INTERFACE PUBLIC RelativeMoveBuilder EXTENDS __System.IQueryInterface

METHOD PUBLIC Acceleration : RelativeMoveBuilder
VAR_INPUT
	value : LREAL;
END_VAR
END_METHOD

METHOD PUBLIC BufferMode : RelativeMoveBuilder
VAR_INPUT
	mode : MotionBufferMode;
END_VAR
END_METHOD

METHOD PUBLIC BuildMoveAdditiveCommand : MotionCommand
VAR_INPUT
	axis : Axis;
END_VAR
END_METHOD

METHOD PUBLIC BuildMoveRelativeCommand : MotionCommand
VAR_INPUT
	axis : Axis;
END_VAR
END_METHOD

METHOD PUBLIC Deceleration : RelativeMoveBuilder
VAR_INPUT
	value : LREAL;
END_VAR
END_METHOD

METHOD PUBLIC Distance : RelativeMoveBuilder
VAR_INPUT
	value : LREAL;
END_VAR
END_METHOD

METHOD PUBLIC Jerk : RelativeMoveBuilder
VAR_INPUT
	value : LREAL;
END_VAR
END_METHOD

METHOD PUBLIC Velocity : RelativeMoveBuilder
VAR_INPUT
	value : LREAL;
END_VAR
END_METHOD

END_INTERFACE

(* stored: Version 1.1.0.1
   Itf RelativeMoveBuilder: Id {bddc8931-0c19-0eb2-24a5-b0ff1c07fd66}
   Folder Builders: Id {6daf0ca8-bdaf-495b-8bb7-ee7370bef123}
   Folder PropertySetters: Id {1d69e98f-87ac-4f4f-9b60-ecee3ad0fec2}
   Method Acceleration: Id {6f259ded-a150-0d36-15c9-f78bb90a64eb}
   Method BufferMode: Id {ac9b4e6c-172d-09f1-2143-396f9f3b2b02}
   Method BuildMoveAdditiveCommand: Id {737ee63a-5b36-048b-3437-5e67558a0659}
   Method BuildMoveRelativeCommand: Id {a776305e-4062-066f-07bb-2fbb58ff07e6}
   Method Deceleration: Id {0e6e74d6-91d3-0325-3fa7-7efc9eaa2442}
   Method Distance: Id {23a8e663-60a3-0135-03f3-8e7c13c775e1}
   Method Jerk: Id {556e6fc9-f979-01e4-163c-9a912f2eac29}
   Method Velocity: Id {745bd3a9-6e78-0053-3978-064d4ff508e1} *)
